{attribute 'qualified_only'}
VAR_GLOBAL
    stTerm1_EK1100   : ST_EK1100;
    stTerm2_EL6070   : ST_EL6070;
    stTerm3_EL6910   : ST_EL6910;
    stTerm4_EL1918   : ST_EL1918;
    stTerm5_EL1918   : ST_EL1918;
    stTerm6_EL2904   : ST_EL2904;
    stTerm7_EL1809   : ST_EL1809;
    stTerm8_EL1809   : ST_EL1809;
    stTerm9_EL2809   : ST_EL2809;
    stTerm10_EL2809  : ST_EL2809;
    stTerm11_EL3058  : ST_EL3058;
	stTerm13_EL2502  : ST_EL2502;
	stTerm15_EL7201  : ST_EL7201;
	stTerm16_EL7201  : ST_EL7201;
	stTerm17_EL7201  : ST_EL7201;
	stTerm18_EL2904  : ST_EL2904;
    stTerm19_EL1809  : ST_EL1809;
	stTerm21_EL3314  : ST_EL3314;
	stTerm20_EL4022  : ST_EL4022;
	stTerm22_EL6633  : ST_EL6633;

    // Festo VABX EtherCAT manifold - Module 2 valve outputs.
    stFestoModule2_VABX : ST_VABX_A_S_BV_V4A;
	stFestoModule3_VABX : ST_VABX_A_S_BV_V4A;
    stFestoModule4_VABX : ST_VABX_A_S_BV_V4A;
	
	// Keyence vs camera
	
	stVSKeyenceCamera	: ST_VS_Keyence_Camera;
	
    // PROFINET Assignable Status, appended separately to preserve camera DUT.
    // Offline linked PROFINET diagnostics; invalid until valid I/O is received.
    wVisionPnState AT %I* : WORD := 16#FFFF;
    wVisionPnDiag AT %I* : WORD := 16#FFFF;
    udiVisionError0Code AT %I* : UDINT;
    udiVisionError1Code AT %I* : UDINT;
    // Diagnostics for the power terminals and the shared Festo coupler.
    stTerm12_EL9410 : ST_EL9410;
    stTerm14_EL9576 : ST_EL9576;
    stFestoTerminalInfo : ST_Terminal_Info;
END_VAR

(* stored: Version 1.1.0.1, ProductVersion 3.1.4026.18
   GVL GVL_EtherCAT: Id {a064ef7b-02e7-4065-97aa-bbc4c525874c} *)
